INTERFACE IPmlStateMachine

METHOD public GetCurrentMode : E_PmlProtectedUnitMode
VAR_INPUT
END_VAR
END_METHOD

METHOD GetCurrentState : E_PMLState
VAR_INPUT
END_VAR
END_METHOD

METHOD PmlModeCommand : BOOL
VAR_INPUT
END_VAR
END_METHOD

METHOD PmlStateCommand : bool
VAR_INPUT
	Command : E_PMLCommand;
END_VAR
END_METHOD

METHOD SetStateComplete : BOOL
VAR_INPUT
END_VAR
END_METHOD

END_INTERFACE

(* stored: Version 1.1.0.1, ProductVersion 3.1.4024.12
   Itf IPmlStateMachine: Id {a572c756-2ee2-4617-b1ba-a370e2347b9e}
   Method GetCurrentMode: Id {30cd7fb2-9a81-454b-9afd-826c85901336}
   Method GetCurrentState: Id {8896b180-4065-4462-9182-dfc33f7be59c}
   Method PmlModeCommand: Id {e47f0040-a872-4910-963e-7f43c8de5a43}
   Method PmlStateCommand: Id {f841f4da-d94f-47fd-a3c7-c8897a849506}
   Method SetStateComplete: Id {5723ee2f-d368-4970-a6c6-2e134230c395} *)
